// TIA Portal V16 export
// export: Created 2022-02-28T20:45:44.0591983Z, ExportSetting WithDefaults, DisplayName Totally Integrated Automation Portal, DisplayVersion V16, DisplayName TIA Portal Version Control Interface, DisplayVersion V16, DisplayName TIA Portal Openness, DisplayVersion V16, DisplayName STEP 7 Professional, DisplayVersion V16, DisplayName STEP 7 Safety, DisplayVersion V16, DisplayName WinCC Advanced, DisplayVersion V16
FUNCTION "01_Mapeo_Entradas" : Void   // FC1, LAD
{ S7_Optimized_Access := 'TRUE' }
VERSION : 0.1
// stored: AutoNumber true, IsIECCheckEnabled false, SetENOAutomatically false, UDAEnableTagReadback false
BEGIN

REGION Network 1: Entradas Fisicas Pistilos
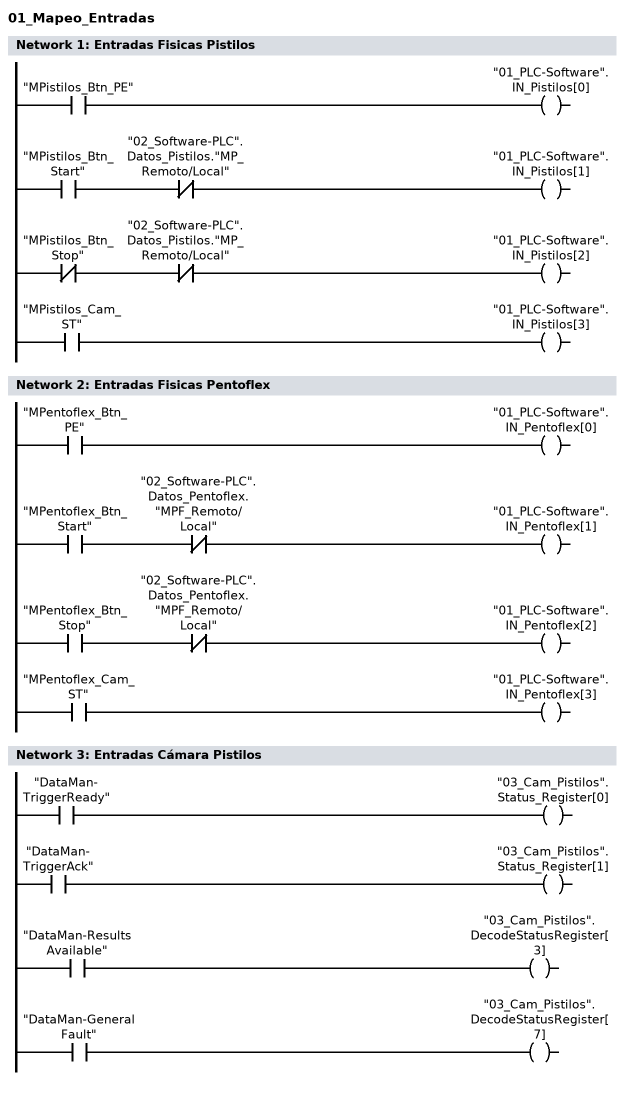
   RUNG wire#powerrail
      Contact( "MPistilos_Btn_PE" )
      Coil( "01_PLC-Software".IN_Pistilos[0] )
   END_RUNG
   RUNG wire#powerrail
      Contact( "MPistilos_Btn_Start" )
      I_Contact( "02_Software-PLC".Datos_Pistilos."MP_Remoto/Local" )
      Coil( "01_PLC-Software".IN_Pistilos[1] )
   END_RUNG
   RUNG wire#powerrail
      I_Contact( "MPistilos_Btn_Stop" )
      I_Contact( "02_Software-PLC".Datos_Pistilos."MP_Remoto/Local" )
      Coil( "01_PLC-Software".IN_Pistilos[2] )
   END_RUNG
   RUNG wire#powerrail
      Contact( "MPistilos_Cam_ST" )
      Coil( "01_PLC-Software".IN_Pistilos[3] )
   END_RUNG
   // the same network as SCL:
   "01_PLC-Software".IN_Pistilos[0] := "MPistilos_Btn_PE";
   "01_PLC-Software".IN_Pistilos[1] := "MPistilos_Btn_Start" AND NOT "02_Software-PLC".Datos_Pistilos."MP_Remoto/Local";
   "01_PLC-Software".IN_Pistilos[2] := NOT "MPistilos_Btn_Stop" AND NOT "02_Software-PLC".Datos_Pistilos."MP_Remoto/Local";
   "01_PLC-Software".IN_Pistilos[3] := "MPistilos_Cam_ST";
END_REGION

REGION Network 2: Entradas Fisicas Pentoflex
   RUNG wire#powerrail
      Contact( "MPentoflex_Btn_PE" )
      Coil( "01_PLC-Software".IN_Pentoflex[0] )
   END_RUNG
   RUNG wire#powerrail
      Contact( "MPentoflex_Btn_Start" )
      I_Contact( "02_Software-PLC".Datos_Pentoflex."MPF_Remoto/Local" )
      Coil( "01_PLC-Software".IN_Pentoflex[1] )
   END_RUNG
   RUNG wire#powerrail
      Contact( "MPentoflex_Btn_Stop" )
      I_Contact( "02_Software-PLC".Datos_Pentoflex."MPF_Remoto/Local" )
      Coil( "01_PLC-Software".IN_Pentoflex[2] )
   END_RUNG
   RUNG wire#powerrail
      Contact( "MPentoflex_Cam_ST" )
      Coil( "01_PLC-Software".IN_Pentoflex[3] )
   END_RUNG
   // the same network as SCL:
   "01_PLC-Software".IN_Pentoflex[0] := "MPentoflex_Btn_PE";
   "01_PLC-Software".IN_Pentoflex[1] := "MPentoflex_Btn_Start" AND NOT "02_Software-PLC".Datos_Pentoflex."MPF_Remoto/Local";
   "01_PLC-Software".IN_Pentoflex[2] := "MPentoflex_Btn_Stop" AND NOT "02_Software-PLC".Datos_Pentoflex."MPF_Remoto/Local";
   "01_PLC-Software".IN_Pentoflex[3] := "MPentoflex_Cam_ST";
END_REGION

REGION Network 3: Entradas Cámara Pistilos
   RUNG wire#powerrail
      Contact( "DataMan-TriggerReady" )
      Coil( "03_Cam_Pistilos".Status_Register[0] )
   END_RUNG
   RUNG wire#powerrail
      Contact( "DataMan-TriggerAck" )
      Coil( "03_Cam_Pistilos".Status_Register[1] )
   END_RUNG
   RUNG wire#powerrail
      Contact( "DataMan-Results Available" )
      Coil( "03_Cam_Pistilos".DecodeStatusRegister[3] )
   END_RUNG
   RUNG wire#powerrail
      Contact( "DataMan-General Fault" )
      Coil( "03_Cam_Pistilos".DecodeStatusRegister[7] )
   END_RUNG
   // the same network as SCL:
   "03_Cam_Pistilos".Status_Register[0] := "DataMan-TriggerReady";
   "03_Cam_Pistilos".Status_Register[1] := "DataMan-TriggerAck";
   "03_Cam_Pistilos".DecodeStatusRegister[3] := "DataMan-Results Available";
   "03_Cam_Pistilos".DecodeStatusRegister[7] := "DataMan-General Fault";
END_REGION

REGION Network 4: Entradas
END_REGION
END_FUNCTION
